// TIA Portal V21 export
// export: Created 2000-01-01T00:00:00.0000000Z, ExportSetting None
TYPE "UDT_Motor"
TITLE = 电机数据结构
// 电机数据 UDT：包含转速反馈、运行状态、故障标志，配合 DB_Motor 使用。
   STRUCT
      Speed { ExternalWritable := 'False'} : Real;   // 电机当前转速反馈值（单位：rpm）
      Run { ExternalWritable := 'False'} : Bool;   // 电机正在运行（起保停输出反馈位）
      Fault { ExternalWritable := 'False'} : Bool;   // 电机故障标志（保留位，由外部诊断置位）
   END_STRUCT;
END_TYPE
